// SIMATIC S7-200 project (STEP 7-Micro/WIN), CPU 221 REL 01.10

ORGANIZATION_BLOCK 主程序:OB1
TITLE=程序注释
BEGIN
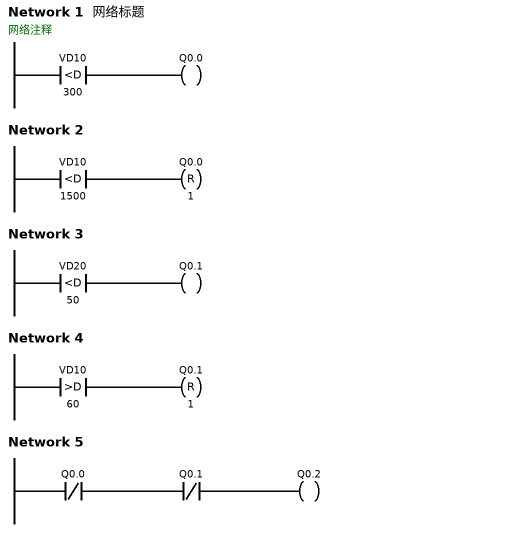
Network 1 // 网络标题
// 网络注释
// (network saved uncompiled; LAD cells follow)
// row 0: c0 -|<D|- VD10, 300  c1 -( ) Q0.0
Network 2
// (network saved uncompiled; LAD cells follow)
// row 0: c0 -|<D|- VD10, 1500  c1 -(R) Q0.0, 1
Network 3
// (network saved uncompiled; LAD cells follow)
// row 0: c0 -|<D|- VD20, 50  c1 -( ) Q0.1
Network 4
// (network saved uncompiled; LAD cells follow)
// row 0: c0 -|>D|- VD10, 60  c1 -(R) Q0.1, 1
Network 5
// (network saved uncompiled; LAD cells follow)
// row 0: c0 -|/|- Q0.0  c1 -|/|- Q0.1  c2 -( ) Q0.2
END_ORGANIZATION_BLOCK
